Fanuc KAREL source: ks00045.KL

-- PROVISIONAL review KL for V1013-1; original PC SHA256 2a0be41d0c085ec6b41f4a934c96f9e23d231b8d08d54ac0c9eeb483f566b11a
-- Incomplete behavior may be omitted. Consult companion uncertainty JSON. Do not deploy.
PROGRAM KS00045
%NOLOCKGROUP
BEGIN
  -- UNRESOLVED_PC offsets 5-13; opcodes 3F,75
  -- UNRESOLVED_PC offsets 18-27; opcodes 3F,75
  -- UNRESOLVED_PC offsets 32-46; opcodes 22,22,1E
  -- UNRESOLVED_PC offsets 51-55; opcodes 7F
END KS00045
